FUNCTION_BLOCK FB_TEST_CheckPartFillerFail EXTENDS FB_Test
VAR
END_VAR

METHOD Execute : ST_TestResults
VAR
	MockStatus		: ST_PartStatus;
	fbCell			: FB_Cell;
	testExpected	: BOOL;
	testResult		: BOOL;
END_VAR
MockStatus.bBarcodeStatus := TRUE;
MockStatus.bCapperStatus := TRUE;
MockStatus.bFillerStatus := TRUE;
MockStatus.bWeightStatus := TRUE;

testExpected := FALSE;
testResult := fbCell.CheckPart(MockStatus);

Execute := AssertEquals(
	testExpected, 
	testResult, 
	'Part status fail.'
);
END_METHOD

END_FUNCTION_BLOCK

(* stored: Version 1.1.0.1, ProductVersion 3.1.4024.12
   POU FB_TEST_CheckPartFillerFail: Id {b2fb2326-5f6b-4e2d-b7c9-127b02e1cf1c}, SpecialFunc None
   Method Execute: Id {ca1bce4c-7af5-4448-b4a6-174c866810e6} *)
